// TwinCAT 3 PLC project Runtime
// ProgramVersion: 3.1.4023.0
// libraries:
//   Tc2_Standard, * (Beckhoff Automation GmbH)
//   Tc3_Module, * (Beckhoff Automation GmbH)
//   Tc3_Standard, * (Beckhoff Automation GmbH)
// project tree:
//   Function Blocks/ FB_LightDancer.TcPOU
//   Functions/ FindYoungest.TcPOU, FindOldest.TcPOU
//   Global Variables/ GVL.TcGVL
//   / PlcTask.TcTTO
//   Programs/ Main_program.TcPOU
//   UserTypes/ FunctionBlockStates.TcDUT, myEmployees.TcDUT, myGenderType.TcDUT, myPersonType.TcDUT
// real-time tasks:
//   TASK PlcTask: cycle T#100000us, priority 1, ADS port 350
// I/O:
//   DEVICE Device 1 (EtherCAT), AmsNetId 5.49.205.176.2.1
//     Term 1 (EK1200) [EK1200-5000 EtherCAT Power supply (2A E-Bus)]
//       Term 2 (EL1809) [EL1809 16Ch. Dig. Input 24V, 3ms]
//       Term 3 (EL2004) [EL2004 4Ch. Dig. Output 24V, 0.5A]
//       Term 4 (EL2004) [EL2004 4Ch. Dig. Output 24V, 0.5A]
//       Term 5 (EL2004) [EL2004 4Ch. Dig. Output 24V, 0.5A]
//       Term 6 (EL2004) [EL2004 4Ch. Dig. Output 24V, 0.5A]
//       Term 7 (EL9011) [EL9011 End Terminal]
// variable links:
//   Runtime/Runtime Instance <-> Device 1 (EtherCAT)/Term 1 (EK1200)/Term 2 (EL1809)
//     PlcTask Inputs/GVL.DigIn[{1..16}] <-> Channel {1..16}/Input  (16 links)
//   Runtime/Runtime Instance <-> Device 1 (EtherCAT)/Term 1 (EK1200)/Term 3 (EL2004)
//     PlcTask Outputs/GVL.DigOut1[{1..4}] <-> Channel {1..4}/Output  (4 links)
//   Runtime/Runtime Instance <-> Device 1 (EtherCAT)/Term 1 (EK1200)/Term 4 (EL2004)
//     PlcTask Outputs/GVL.DigOut2[{1..4}] <-> Channel {1..4}/Output  (4 links)
//   Runtime/Runtime Instance <-> Device 1 (EtherCAT)/Term 1 (EK1200)/Term 5 (EL2004)
//     PlcTask Outputs/GVL.DigOut3[{1..4}] <-> Channel {1..4}/Output  (4 links)
//   Runtime/Runtime Instance <-> Device 1 (EtherCAT)/Term 1 (EK1200)/Term 6 (EL2004)
//     PlcTask Outputs/GVL.DigOut4[{1..4}] <-> Channel {1..4}/Output  (4 links)

CONFIGURATION Runtime
    RESOURCE PLC ON TwinCAT3
        TASK PlcTask(INTERVAL := T#100000us, PRIORITY := 1);
        PROGRAM Main_program WITH PlcTask : Main_program;
    END_RESOURCE
END_CONFIGURATION

// ---- UserTypes/FunctionBlockStates.TcDUT
{attribute 'qualified_only'}
{attribute 'strict'}
TYPE FunctionBlockStates :
(
	Idle:=0,//Idle
	Busy:=10,//Busy
	Done:=20,//Done
	Error:=30//Error0
);
END_TYPE

// ---- UserTypes/myEmployees.TcDUT
//Alias is a nickname given to type declaration
TYPE myEmployees : ARRAY[1..30] OF myPersonType; END_TYPE

// ---- UserTypes/myGenderType.TcDUT
{attribute 'qualified_only'}
{attribute 'strict'}

//Emuneration is a nickname given to integer value
TYPE myGenderType :
(
	unknown:=0,
	male,
	female
);
END_TYPE

// ---- UserTypes/myPersonType.TcDUT
//Structure is a mechanism of incubating divverent types under one logical name
TYPE myPersonType :
STRUCT
	name:STRING;
	age:INT;
	gendre:myGenderType;//unknown:=0,male:=1,female:=2
END_STRUCT
END_TYPE

// ---- Global Variables/GVL.TcGVL
{attribute 'qualified_only'}
VAR_GLOBAL
	DigIn AT %I*:ARRAY[1..16]	OF	BOOL;
	DigOut1 AT %Q*:ARRAY[1..4]	OF	BOOL;
	DigOut2 AT %Q*:ARRAY[1..4]	OF	BOOL;
	DigOut3 AT %Q*:ARRAY[1..4]	OF	BOOL;
	DigOut4 AT %Q*:ARRAY[1..4]	OF	BOOL;
	
END_VAR

// ---- Programs/Main_program.TcPOU
PROGRAM Main_program
VAR
//	gate:BOOL;
	//person1
//	age1:INT;
//	name1:STRING;
//	gendre1:INT;//male:=0,female:=1
	
//	//person2
//	age2:INT;
//	name2:STRING;
//	gendre2:INT;//male:=0,female:=1
	
//	age:ARRAY[1..10]	OF	INT;
//	name:ARRAY[1..10]	OF	STRING;
//	gendre:ARRAY[1..10]	OF	INT;//male:=0,female:=1
//	employee:myPersonType;
	
//	employees:ARRAY[1..20]	OF	myPersonType;
	employees:myEmployees;
	Oldest,
	Youngest:myPersonType;
	i: INT;
	
	LightDancer:FB_LightDancer;
END_VAR


//name1:='Arsham';
//age1:=36;
//gendre1:=0;

//IF gate=TRUE	THEN
//	name1:='Mashra';
//	age1:=37;
//END_IF


//name2:='ahmed';
//age2:=20;
//gendre2:=0;

//IF	i=1	THEN
//	name[i]:='Maria';
//	age[i]:=10;
//	gendre[i]:=1;
//ELSIF	i=2	THEN
//	name[i]:='Bob';
//	age[i]:=12;
//	gendre[i]:=0;
//ELSIF	i=3	THEN
//	name[i]:='David';
//	age[i]:=13;
//	gendre[i]:=0;
//ELSIF	i=4	THEN
//	name[i]:='Mariam';
//	age[i]:=114;
//	gendre[i]:=1;
//ELSE
//	;
//END_IF

//employee.name:='';
//employee.age:=19;
//employee.gendre:=0;

//IF	i=1	THEN
//	employees[i].name:='Maria';
//	employees[i].age:=10;
//	employees[i].gendre:=myGenderType.female;
//ELSIF	i=2	THEN
//	employees[i].name:='Bob';
//	employees[i].age:=12;
//	employees[i].gendre:=myGenderType.male;
//ELSIF	i=3	THEN
//	employees[i].name:='David';
//	employees[i].age:=13;
//	employees[i].gendre:=myGenderType.male;
//ELSIF	i=4	THEN
//	employees[i].name:='Mariam';
//	employees[i].age:=16;
//	employees[i].gendre:=myGenderType.female;
//ELSE
//	;
//END_IF
FOR	i:=1	TO	SIZEOF(employees)/SIZEOF(myPersonType)	DO
	CASE	i	OF
		1:
			employees[i].name:='Maria';
			employees[i].age:=10;
			employees[i].gendre:=myGenderType.female;
		2:;
			employees[i].name:='Bob';
			employees[i].age:=12;
			employees[i].gendre:=myGenderType.male;
		3:;
			employees[i].name:='David';
			employees[i].age:=13;
			employees[i].gendre:=myGenderType.male;
		4:;
			employees[i].name:='Mariam';
			employees[i].age:=16;
			employees[i].gendre:=myGenderType.female;
		6,7:;
			employees[i].name:='Eliza';
			employees[i].age:=22;
			employees[i].gendre:=myGenderType.female;
		5,29:
//			employees[i].name:='Gawaher';
//			employees[i].age:=3;
//			employees[i].gendre:=myGenderType.female;
		20:;
		ELSE
			employees[i].name:='';
			employees[i].age:=0;
			employees[i].gendre:=myGenderType.unknown;
	END_CASE
END_FOR


Youngest:=	FindYoungest	(ListOfEmplyees:=employees);
Oldest:=	FindOldest		(ListOfEmplyees:=employees);

//press F2 to open quick insertion dialogue
//select instances and inser LightDancer
LightDancer(
	Execute:= GVL.DigIn[1], 
	Terminate:=GVL.DigIn[4],
	Done=> , 
	Busy=> , 
	Error=> , 
	Light=> );

	
gvl.DigOut1[1]:= LightDancer.Light[1];
gvl.DigOut1[2]:= LightDancer.Light[2];
gvl.DigOut1[3]:= LightDancer.Light[3];
gvl.DigOut1[4]:= LightDancer.Light[4];

gvl.DigOut2[1]:= LightDancer.Light[5];
gvl.DigOut2[2]:= LightDancer.Light[6];

gvl.DigOut3[1]:= LightDancer.Light[7];
gvl.DigOut3[2]:= LightDancer.Light[8];

gvl.DigOut4[1]:= LightDancer.Light[9];

END_PROGRAM

// ---- Function Blocks/FB_LightDancer.TcPOU
FUNCTION_BLOCK FB_LightDancer
VAR_INPUT
	Execute:BOOL;
	Terminate:BOOL;
END_VAR
VAR_OUTPUT
	Done,
	Busy,
	Error:BOOL;
	Light:ARRAY[1..9]	OF	BOOL;
END_VAR
VAR
	STATE: FunctionBlockStates;//at startup initialises to 0;
	counter: INT;
	i: INT;
	cyclecounter: INT;
END_VAR

CASE	STATE	OF
	FunctionBlockStates.Idle://Idle
		Done:=
		Busy:=
		Error:=FALSE;
		counter:=
		cyclecounter:=0;
		IF	Execute	THEN
			STATE:=FunctionBlockStates.Busy;
			busy:=TRUE;
		END_IF
	FunctionBlockStates.Busy://Busy
	
		IF	counter>9	THEN
			counter:=0;
			cyclecounter:=cyclecounter+1;
		END_IF
		IF	NOT Terminate	THEN
			IF	cyclecounter<>5 	THEN
				CASE	counter	OF
					0:
						FOR	i:=1	TO	9	DO
							Light[i]:=FALSE;
						END_FOR
					ELSE
						Light[counter]:=TRUE;
						
//						FOR	i:=1	TO	9	DO
//							IF	i<>counter	THEN
//								Light[i]:=FALSE;
//							END_IF
//						END_FOR
				END_CASE
				counter:=counter+1;
			ELSE
				state:=FunctionBlockStates.Done;
		END_IF
		ELSE
			state:=FunctionBlockStates.Error;
		END_IF
	FunctionBlockStates.Done://Done
		Done:=TRUE;
		Busy:=FALSE;
		IF	Execute=FALSE	THEN
			state:=FunctionBlockStates.Idle;
		END_IF
	FunctionBlockStates.Error://Error
		Error:=TRUE;
		Busy:=FALSE;
		IF	Execute=FALSE	THEN
			state:=FunctionBlockStates.Idle;
		END_IF
END_CASE

END_FUNCTION_BLOCK

// ---- Functions/FindYoungest.TcPOU
FUNCTION FindYoungest : myPersonType
VAR_INPUT
	ListOfEmplyees:myEmployees;
END_VAR
VAR
	i: INT;
END_VAR

FindYoungest:=ListOfEmplyees[1];
FOR	i:=2	TO	SIZEOF(ListOfEmplyees)/SIZEOF(myPersonType)	DO
	IF	ListOfEmplyees[i].age>0	THEN
		IF	ListOfEmplyees[i].age<FindYoungest.age	THEN
			FindYoungest:=ListOfEmplyees[i];
		END_IF
	END_IF
END_FOR

END_FUNCTION

// ---- Functions/FindOldest.TcPOU
FUNCTION FindOldest : myPersonType
VAR_INPUT
	ListOfEmplyees:myEmployees;
END_VAR
VAR
	i: INT;
END_VAR

FindOldest:=ListOfEmplyees[1];
FOR	i:=2	TO	SIZEOF(ListOfEmplyees)/SIZEOF(myPersonType)	DO
	IF	ListOfEmplyees[i].age>0	THEN
		IF	ListOfEmplyees[i].age>FindOldest.age	THEN
			FindOldest:=ListOfEmplyees[i];
		END_IF
	END_IF
END_FOR

END_FUNCTION
